INTERFACE I_AnimalFamily

END_INTERFACE

(* stored: Version 1.1.0.1, ProductVersion 3.1.4024.16
   Itf I_AnimalFamily: Id {0208a277-f525-4eb4-bd48-e03741525f8f} *)
